Fanuc KAREL source: NC0036.KL

-- PROVISIONAL review KL for V940-1; original PC SHA256 507a1f99e9eba70f9a116fe90405c9ed10bf59d51b2036426e8152e708e860f8
-- Incomplete behavior may be omitted. Consult companion uncertainty JSON. Do not deploy.
PROGRAM NC0036
%NOLOCKGROUP
-- UNRESOLVED_LOCAL_POOL 1 cells at code offset 3; source declarations unknown
-- DIRECT_LOCAL_WORD_ACCESS alone does not prove INTEGER, REAL, or BOOLEAN
BEGIN
  -- UNRESOLVED_PC offsets 0-8; opcodes 2B,2C,7B
  -- UNRESOLVED_PC offsets 13-20; opcodes 9D,23
  -- UNRESOLVED_PC offsets 25-42; opcodes 21,40,41,42
  -- UNRESOLVED_PC offsets 47-81; opcodes 21,2E,52,23,7A,40,41,42
  -- UNRESOLVED_PC offsets 86-110; opcodes 21,2E,52,23,7A,43
  -- UNRESOLVED_PC offsets 115-132; opcodes 21,40,41,42
  -- UNRESOLVED_PC offsets 137-171; opcodes 21,2E,52,23,7A,40,41,42
  -- UNRESOLVED_PC offsets 176-200; opcodes 21,2E,52,23,7A,43
  -- UNRESOLVED_PC offsets 205-222; opcodes 21,40,41,42
  -- UNRESOLVED_PC offsets 227-261; opcodes 21,2E,52,23,7A,40,41,42
  -- UNRESOLVED_PC offsets 266-290; opcodes 21,2E,52,23,7A,43
  -- UNRESOLVED_PC offsets 295-312; opcodes 21,40,41,42
  -- UNRESOLVED_PC offsets 317-351; opcodes 21,2E,52,23,7A,40,41,42
  -- UNRESOLVED_PC offsets 356-380; opcodes 21,2E,52,23,7A,43
  -- UNRESOLVED_PC offsets 385-402; opcodes 21,40,41,42
  -- UNRESOLVED_PC offsets 407-441; opcodes 21,2E,52,23,7A,40,41,42
  -- UNRESOLVED_PC offsets 446-470; opcodes 21,2E,52,23,7A,43
  -- UNRESOLVED_PC offsets 475-492; opcodes 21,40,41,42
  -- UNRESOLVED_PC offsets 497-531; opcodes 21,2E,52,23,7A,40,41,42
  -- UNRESOLVED_PC offsets 536-560; opcodes 21,2E,52,23,7A,43
  -- UNRESOLVED_PC offsets 565-582; opcodes 21,40,41,42
  -- UNRESOLVED_PC offsets 587-621; opcodes 21,2E,52,23,7A,40,41,42
  -- UNRESOLVED_PC offsets 626-650; opcodes 21,2E,52,23,7A,43
  -- UNRESOLVED_PC offsets 655-672; opcodes 21,40,41,42
  -- UNRESOLVED_PC offsets 677-711; opcodes 21,2E,52,23,7A,40,41,42
  -- UNRESOLVED_PC offsets 716-740; opcodes 21,2E,52,23,7A,43
  -- UNRESOLVED_PC offsets 745-759; opcodes 21,9D,52,23
  -- UNRESOLVED_PC offsets 804-808; opcodes 7F
  -- UNRESOLVED_PC offsets 813-817; opcodes 27,AA
  -- UNRESOLVED_PC offsets 822-826; opcodes 7F
END NC0036
